// SIMATIC S7-200 SMART project (STEP 7-Micro/WIN SMART), CPU SR40

ORGANIZATION_BLOCK 主程序:OB1
TITLE=程序注释
BEGIN
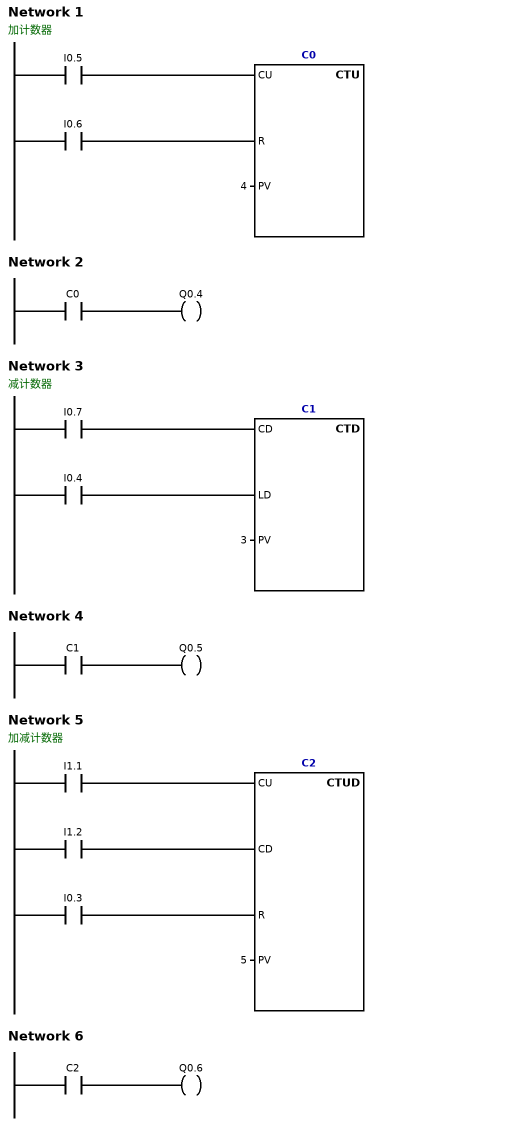
Network 1
// 加计数器
LD     I0.5
LD     I0.6
CTU    C0, 4
Network 2
LD     C0
=      Q0.4
Network 3
// 减计数器
LD     I0.7
LD     I0.4
CTD    C1, 3
Network 4
LD     C1
=      Q0.5
Network 5
// 加减计数器
LD     I1.1
LD     I1.2
LD     I0.3
CTUD   C2, 5
Network 6
LD     C2
=      Q0.6
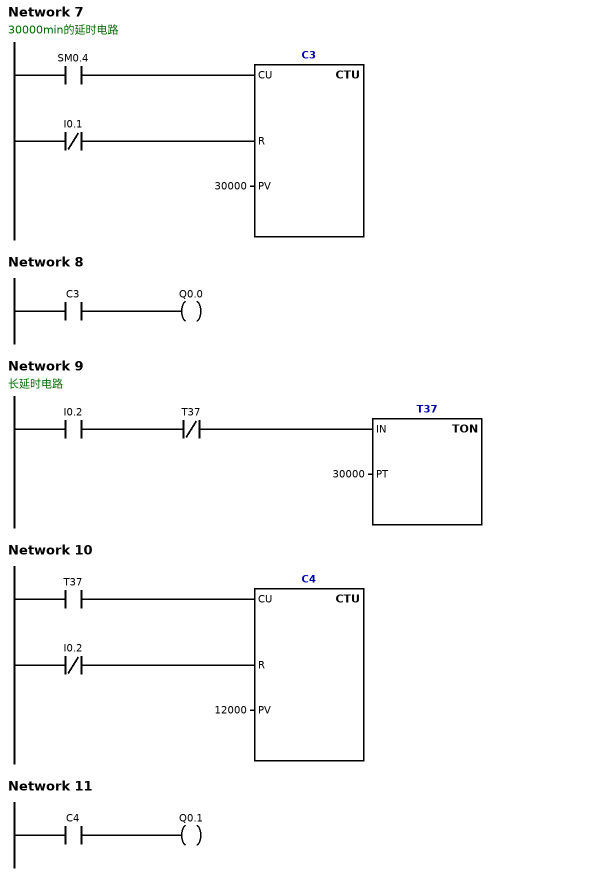
Network 7
// 30000min的延时电路
LD     SM0.4
LDN    I0.1
CTU    C3, 30000
Network 8
LD     C3
=      Q0.0
Network 9
// 长延时电路
LD     I0.2
AN     T37
TON    T37, 30000
Network 10
LD     T37
LDN    I0.2
CTU    C4, 12000
Network 11
LD     C4
=      Q0.1
END_ORGANIZATION_BLOCK
